FUNCTION_BLOCK E_CYCLE
  (* Version 1.0, 2005-06-24, Goran Cengic, Chalmers, Released under the GNU General Public License (GLP). *)
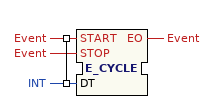
  EVENT_INPUT
    START WITH DT;
    STOP;
  END_EVENT
  EVENT_OUTPUT
    EO;
  END_EVENT
  VAR_INPUT
    DT : INT;
  END_VAR
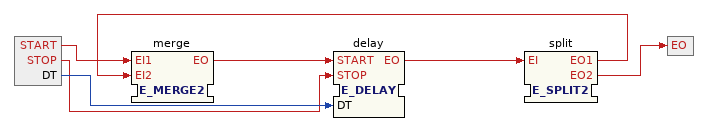
  FBS
    merge : E_MERGE2;
    delay : E_DELAY;
    split : E_SPLIT2;
  END_FBS
  EVENT_CONNECTIONS
    START TO merge.EI1;
    merge.EO TO delay.START;
    delay.EO TO split.EI;
    split.EO1 TO merge.EI2;
    split.EO2 TO EO;
    STOP TO delay.STOP;
  END_CONNECTIONS
  DATA_CONNECTIONS
    DT TO delay.DT;
  END_CONNECTIONS
END_FUNCTION_BLOCK
